(* PLC project liner_cyclic.project, CODESYS CODESYS V3.5 SP17 Patch 3 *)
(* stored: creationDateTime 1970-01-01T00:00:00, modificationDateTime 1970-01-01T00:00:00 *)

PROGRAM ServoControl
  VAR
    fbPower : MC_Power;
    fbStop : MC_Stop;
    fbReset : MC_Reset;
    fbReadActualPosition : MC_ReadActualPosition;
    bRegulatorOn : BOOL := FALSE;
    bDriveStart : BOOL := FALSE;
    btn : BOOL := FALSE;
    bReset : BOOL;
    bStop : BOOL;
    fbLinearSensorHandle : LinearSensorHandle;  (* /////////////////////////////////////// *)
    mm : REAL;
    Busy : BOOL;
    Error : BOOL;
    fbReadFBError : SMC_ReadFBError;  (* //////////////////SMC_ReadFBError////////////////////// *)
    ReadFBErrorValid : BOOL;
    ReadFBErrorBusy : BOOL;
    ReadFBErrorError : BOOL;
    ReadFBErrorErrorID : SMC_Error;
    ReadFBErrorTimestamp : TIME;
    ton : TON;
    tof : TOF;
    ET_TON : TIME;
    ET_TOF : TIME;
    bflag : BOOL := FALSE;
    rs : rs;
    fbHalt : MC_Halt;
    bfbHaltOn : BOOL;
    lrfbHaltDeceleration : LREAL := 0.01;
    bfbHaltDone : BOOL;
    fbJog : MC_Jog;
    fbJog_0 : MC_Jog;
    lrfbJogVelocity : LREAL := 100;
    lrfbJogAcceleration : LREAL := 100;
    lrfbJogDeceleration : LREAL := 1000;
    lrfbJogJerk : LREAL := 10;
    bfbJogBusy : BOOL;
    sp : REAL;  (* уставка *)
    fbReadStatus : MC_ReadStatus;  (* /////////////////////fbReadStatus/////////////////////////// *)
    bfbFollowVelocityBusy : BOOL;
    bClearFBError : BOOL;
    ClearFBError_r_trig : R_TRIG;
    Y_MIN : REAL;
    Y_MAX : REAL;
    bStandStill : BOOL;
    r_trig1 : R_TRIG;
    rMin : REAL;
    rMax : REAL;
    lrCurrentPosition : LREAL;  (* /////////////fbReadActualPosition///////////////////// *)
    fbGenSQR : OSCAT_BASIC.GEN_SQR;  (* /////////////fbGenSQR///////////////////// *)
    fbGenSQR_Q : BOOL;
    fbGenSQR_OUT : REAL;
    fbFreq_Measure : FREQ_MEASURE;  (* /////////////fbFreq_Measure/////////////// *)
    fbFreq_Measure_reset : BOOL;
    fbFreq_Measure_current_freq : REAL;
    fbFreq_Measure_valid : BOOL;
    _PT : TIME;
    _AM : REAL;
    _OS : REAL;
    _DC : REAL;
    _DL : REAL;
    GenSignalOUT_TMP : REAL;
    bSelect_gen_signal_btn : BOOL := FALSE;  (* 0 - SIN, 1 - SQR *)
    fbGen_SIN : OSCAT_BASIC.GEN_SIN;  (* /////////////fbGen_SIN//////////////////////////// *)
    fbGen_SIN_Q : BOOL;
    OUT : REAL;
    offset_1 : REAL;
    out_after_offset : REAL;
    fbMoveRelative : MC_MoveRelative;  (* ////MoveRelative///////////////// *)
    bExecuteMR : BOOL;
    lrDistanceMR_PLUS : LREAL;
    lrVelocityMR : LREAL;
    lrAccelerationMR : LREAL;
    lrDecelerationMR : LREAL;
    bPuskMR : BOOL;
    fbMoveRelative2 : MC_MoveRelative;
    lrDistanceMR_MINUS : LREAL;
    PLUS : LREAL;
    MINUS : LREAL;
    fbFollowPosition : SMC_FollowPosition;  (* ////SMC_FollowPosition//////// *)
    bExecuteFP : BOOL := FALSE;
    lrfSetPositionFP : LREAL;
    lrTMP_PLUS_MINUS : LREAL;
    r_trig123 : R_TRIG;
    TON_0 : TON;  (* /////////////////////// *)
    TON_0_ET : TIME;
    fbLIN_TRAFO_0 : LIN_TRAFO;
    units : REAL;
    mm_tmp : REAL;
    out_FORCE_TMP : REAL;
    rSetMaxPrednagruzka_USTAVKA : REAL := 500;  (* В Н(Ньютонах) *)
    bBtnPrednagruzkaON : BOOL;  (* Включить режим преднагрузка *)
    rSetIncPrednagruzka_USTAVKA : REAL := 10;  (* Инкремент нагружения *)
    RS_2 : RS;
    ustavka_HERZ : REAL := 1;  (* //////////////////////////////////////////////////////////////////////// *)
    pt_test : TIME;
    ustavka_H : REAL;
  END_VAR

            //Выставить только AM - амплитуду из расчета = если нужно от 0 до 10 , то ставим AM = 20, OS = 0, DL = 0;
//с offset: если поставить AM = 30, offset_1 = 30 => rout_after_offset от 15 до 45
Errors();
Halt();
Jog();
MainAlgorithm();
Power();
Reset();
Status();
Stop();












	





	

	
	


	








	



          

ACTION Power:
                IF Y_Axis.bCommunication THEN
// Функциональный блок влючения
fbPower(
Axis:= Y_Axis ,
Enable:= TRUE,
bRegulatorOn:= bRegulatorOn,
bDriveStart:= bDriveStart,
Status=> ,
bRegulatorRealState=> ,
bDriveStartRealState=> ,
Busy=> Busy,
Error=> Error,
ErrorID=> );
END_IF

r_trig1(CLK := GVL.bAlarm OR SafetyChain.bHomePosition);
IF btn AND (NOT GVL.bAlarm) AND (NOT SafetyChain.bHomePosition) THEN
	bRegulatorOn := TRUE;
	bDriveStart := TRUE;
	ELSIF (NOT btn) OR (GVL.bAlarm) OR (SafetyChain.bHomePosition) THEN
	bRegulatorOn := FALSE;
	bDriveStart := FALSE;
	
END_IF

IF r_trig1.Q THEN
	btn := FALSE;
END_IF


IF fbPower.Status THEN
	//bMoveRelativeON := TRUE;
	//bMoveAbsoluteON := TRUE;
	ELSE
	//bMoveRelativeON := FALSE;
	//bMoveAbsoluteON := FALSE;
END_IF
              
END_ACTION

ACTION Stop:
                //Функциональный блок останова
fbStop(
Axis:= Y_Axis,
Execute:= bStop,
Deceleration:= ,
Jerk:= ,
Done=> ,
Busy=> ,
Error=> ,
ErrorID=> );
              
END_ACTION

ACTION Reset:
                
	rs(SET := GVL.breset_btn, RESET1 := tof.Q);
	ton(IN := ReadFBErrorError AND rs.Q1, PT := T#0.5S , ET => ET_TON);
	tof(IN := bFlag ,PT := T#0.5S, ET =>ET_TOF);
	IF ton.Q THEN
		btn := FALSE;
		bReset := TRUE;
		bFlag := TRUE;
	END_IF
	IF tof.Q THEN
		btn := TRUE;
		bReset := FALSE;
		bFlag := FALSE;
		gvl.breset_btn := FALSE;
END_IF

// Фунциональный блок RESET
fbReset (
Axis:= Y_Axis ,
Execute:= bReset,
Done=> ,
Busy=> ,
Error=> ,
ErrorID=> );
              
END_ACTION

ACTION Jog:
                IF NOT ReadFBErrorError AND fbPower.Status THEN



fbJog(
	Axis:= Y_Axis, 
	JogForward:= GVL.bfbJogJogForward,   // против часовой (+ ServoControl.LrPosition_readActPos)  ВНИЗ
	JogBackward:= GVL.bfbJogJogBackward, // по часовой (- ServoControl.LrPosition_readActPos) ВВЕРХ
	Velocity:= lrfbJogVelocity, 
	Acceleration:= lrfbJogAcceleration, 
	Deceleration:= lrfbJogDeceleration, 
	Jerk:= lrfbJogJerk, 
	Busy=> bfbJogBusy, 
	CommandAborted=> , 
	Error=> , 
	ErrorId=> );
	
	

	END_IF

	
	
              
END_ACTION

ACTION MainAlgorithm:
                	(*
	// Движение вниз циклично
	fbMoveRelative(
	Axis:= Y_Axis, 
	Execute:= (bExecuteMR OR fbGenSQR_Q) AND bPuskMR, 
	Distance:= lrDistanceMR_PLUS, 
	Velocity:= lrVelocityMR, 
	Acceleration:= lrAccelerationMR, 
	Deceleration:= lrDecelerationMR, 
	Jerk:= , 
	BufferMode:= , 
	Done=> , 
	Busy=> , 
	Active=> , 
	CommandAborted=> , 
	Error=> , 
	ErrorID=> );
	
	// Движение вверх циклично
	fbMoveRelative2(
	Axis:= Y_Axis, 
	Execute:= (bExecuteMR OR NOT fbGenSQR_Q) AND bPuskMR, 
	Distance:= lrDistanceMR_MINUS, 
	Velocity:= lrVelocityMR, 
	Acceleration:= lrAccelerationMR, 
	Deceleration:= lrDecelerationMR, 
	Jerk:= , 
	BufferMode:= , 
	Done=> , 
	Busy=> , 
	Active=> , 
	CommandAborted=> , 
	Error=> , 
	ErrorID=> );
	*)

	// Движение согласно закону (Квадратично/Синусоидально)
	fbFollowPosition(
	Axis:= Y_Axis, 
	bExecute:= bExecuteFP, 
	//fSetPosition:= lrfSetPositionFP + lrTMP_PLUS_MINUS, 
	fSetPosition:= lrfSetPositionFP + OUT,  //текущая позиция + отклонение согласно квадратично/синусоидальному закону 
	bBusy=> , 
	bCommandAborted=> , 
	bError=> , 
	iErrorID=> );
	
	//При нажатии на кнопку "btn" фиксируем текущую позицию
	r_trig123(CLK := ServoControl.btn);
	IF r_trig123.Q THEN
	lrfSetPositionFP := lrCurrentPosition;    	
	END_IF
	
	//Текущая позиция
	fbReadActualPosition(
	Axis:= Y_Axis, 
	Enable:= TRUE, 
	Valid=> , 
	Busy=> , 
	Error=> , 
	ErrorID=> , 
	Position=> lrCurrentPosition);

	//bSelect_gen_signal_btn - 0 -> SIN, bSelect_gen_signal_btn - 1 -> SQR 
	IF bSelect_gen_signal_btn THEN
	///////КВАДРАТ/////////////////
	fbGenSQR(
	PT:= _PT, 
	AM:= _AM, 
	OS:= _OS, 
	DC:= _DC, 
	DL:= _DL, 
	Q=> fbGenSQR_Q, 
	Out=> OUT);
	
	IF fbGenSQR_Q = TRUE THEN
		GenSignalOUT_TMP := OUT;
		lrDistanceMR_PLUS := PLUS;
		lrTMP_PLUS_MINUS := PLUS;
	END_IF
	
	IF fbGenSQR_Q = FALSE THEN
		GenSignalOUT_TMP := 0;
		lrDistanceMR_MINUS := MINUS;
		lrTMP_PLUS_MINUS := MINUS;
	END_IF
	
	fbFreq_Measure(
	IN:= fbGenSQR_Q, 
	PERIODS:= 1, 
	RESET:= fbFreq_Measure_reset, 
	OUT=> fbFreq_Measure_current_freq, 
	VALID=> fbFreq_Measure_valid);
	ELSE
	//////////////СИНУС////////////////////	
	fbGen_SIN(
	PT:= _PT, 
	AM:= _AM, 
	OS:= _OS, 
	DL:= _DL, 
	Q=> fbGen_SIN_Q, 
	Out=> OUT);
		
	IF fbGen_SIN_Q = TRUE THEN
		GenSignalOUT_TMP := OUT;
	END_IF
	
	IF fbGen_SIN_Q = FALSE THEN
		GenSignalOUT_TMP := 0;
	END_IF
	
	//Частота в Гц
	fbFreq_Measure(
	IN:= fbGen_SIN_Q, 
	PERIODS:= 1, 
	RESET:= fbFreq_Measure_reset, 
	OUT=> fbFreq_Measure_current_freq, 
	VALID=> fbFreq_Measure_valid);
	END_IF
	//////////////////////////////////////////////////////////////////////////////
	(*
	out_after_offset := OSCAT_BASIC.OFFSET(
	X:= GenSignalOUT_TMP, 
	O1:= TRUE, 
	O2:= FALSE, 
	O3:= FALSE, 
	O4:= FALSE, 
	D:= FALSE, 
	Offset_1:= offset_1,
	Offset_2:= 0,
	Offset_3:= 0,
	Offset_4:= 0,
	default:= 0);   *)

//Переводим условные единицы в мм
fbLinearSensorHandle(position := GVL.KTSL_Position_1, Calc_position_mm => mm);

//мм в юниты   Заменить mm_tmp на mm
fbLIN_TRAFO_0(
	IN:= mm, 
	IN_MIN:= 0, 
	IN_MAX:= 1000, 
	OUT_MIN:= -1666611.98, 
	OUT_MAX:= -1521270.48, 
	OUT=> units, 
	ERROR=> );

// Преобразование ГЦ во время _PT
_PT := real_TO_TIME(EXPT(ustavka_HERZ, -1) * 1000);

// Задать диапазон отклонения сигнала 
_AM := ustavka_H * 2;





              
END_ACTION

ACTION Status:
                fbReadStatus(
	Axis:= Y_Axis, 
	Enable:= TRUE, 
	Valid=> , 
	Busy=> , 
	Error=> , 
	ErrorID=> , 
	Disabled=> , 
	Errorstop=> , 
	Stopping=> , 
	StandStill=> bStandStill, 
	DiscreteMotion=> , 
	ContinuousMotion=> , 
	SynchronizedMotion=> , 
	Homing=> , 
	ConstantVelocity=> , 
	Accelerating=> , 
	Decelerating=> , 
	FBErrorOccured=> );
	
	
	//DriveStatus := Y_Axis.nAxisState;  // Статус привода
              
END_ACTION

ACTION Errors:
                fbReadFBError(
	Axis:= Y_Axis, 
	bEnable:= TRUE, 
	bValid=> ReadFBErrorValid, 
	bBusy=> ReadFBErrorBusy, 
	bFBError=> ReadFBErrorError, //ОШИБКА ПРИВОДА
	nFBErrorID=> ReadFBErrorErrorID, 
	pbyErrorInstance=> , 
	strErrorInstance=> , 
	tTimeStamp=> ReadFBErrorTimestamp);
	
	ClearFBError_r_trig(CLK := bClearFBError);   // очистка аварий
IF ClearFBError_r_trig.Q THEN
	SMC_ClearFBError(pDrive:= ADR(Y_Axis));
END_IF
              
END_ACTION

ACTION Halt:
                IF NOT ReadFBErrorError AND fbPower.Status THEN
fbHalt(                            // Остановка с регулируемым замедлением  
	Axis:= Y_Axis, 
	Execute:= bfbHaltOn, 
	Deceleration:= lrfbHaltDeceleration, 
	Jerk:= 100, 
	Done=> bfbHaltDone, 
	Busy=> , 
	CommandAborted=> , 
	Error=> , 
	ErrorID=> );
END_IF
              
END_ACTION

ACTION Prednagruzka:
                //IF NOT ReadFBErrorError AND fbPower.Status THEN

	RS_2(SET:= bBtnPrednagruzkaON, RESET1:= out_FORCE_TMP > rSetMaxPrednagruzka_USTAVKA, Q1=> );
fbJog_0(
	Axis:= Y_Axis, 
	JogForward:= RS_2.Q1,   // против часовой (+ ServoControl.LrPosition_readActPos)  ВНИЗ
	JogBackward:= , // по часовой (- ServoControl.LrPosition_readActPos) ВВЕРХ
	Velocity:= lrfbJogVelocity, 
	Acceleration:= lrfbJogAcceleration, 
	Deceleration:= lrfbJogDeceleration, 
	Jerk:= lrfbJogJerk, 
	Busy=> bfbJogBusy, 
	CommandAborted=> , 
	Error=> , 
	ErrorId=> );


	//END_IF

              
END_ACTION
END_PROGRAM
